// Funzione che ritorna TRUE tutti i WORKFLOW sono almeno in uno dei seguenti stati: Disabilitato,Errore,Terminato
FUNCTION TFIsWorkflowDisableOrEndedOrError : BOOL 
VAR_INPUT
	NumWFPresence : UINT;
	WorkFlow : POINTER TO ARRAY[0..MAXWORKFLOW] OF WorkFlow;
END_VAR
VAR
	i: UINT;
END_VAR


FOR i:=0 TO NumWFPresence DO
	IF WorkFlow^[i].Enable = FALSE OR WorkFlow^[i].State = StateWF_END OR WorkFlow^[i].State = StateWF_END THEN
		TFIsWorkflowDisableOrEndedOrError := TRUE;
	ELSE
		TFIsWorkflowDisableOrEndedOrError := FALSE;
		RETURN;
	END_IF
END_FOR

END_FUNCTION

(* stored: Version 1.1.0.1, ProductVersion 3.1.4024.11
   POU TFIsWorkflowDisableOrEndedOrError: Id {7cdab8e6-e6e8-4442-aeed-fee484ff8c82}, SpecialFunc None *)
